FUNCTION_BLOCK RunUnitIndexerMasterCelluarA EXTENDS RunUnitIndexerMaster
VAR_INPUT
	// conveyor related , Fast + Slow = pitch
	ptCommandFast : POINTER TO CommandBlockPos;
	ptCommandSlow : POINTER TO CommandBlockPos;
	ptCommandExtend : POINTER TO CommandBlockPos;
	//Checkpoints
	ptCommandTriggerRaise: POINTER TO CommandBlockPos; //trigger point
	ptCommandCheckRaise : POINTER TO commandBlockPos; //if not all lifter done until then , stop conveyor motion
	ptCommandCheckReach : POINTER TO commandBlockPos;
	//Lifters
	lifters : ARRAY[1..3] OF POINTER TO RunLifterCelluar;
END_VAR
VAR_OUTPUT
END_VAR
VAR
	bFast : BOOL;
	bSlow : BOOL;
	bExtend : BOOL;
	
	nCounter  : INT ;
	allLifterDone : BOOL;
	allLifterReach: BOOL;
END_VAR

//implement state 3

SUPER^(); //run indexer master

//Buffer modes
ptAxisMaster^.ExecuteCommandBlock(ptBlock := ptCommandFast,
	Execute:= bFast,
	Done=>);
ptAxisMaster^.ExecuteCommandBlock(ptBlock := ptCommandSlow,
	Execute:= bSlow,
	Done=>);
ptAxisMaster^.ExecuteCommandBlock(ptBlock := ptCommandExtend,
	Execute:= bExtend,
	Done=>);

allLifterDone := TRUE; //reset
FOR nCounter:=1 TO 3 BY 1 DO
	lifters[nCounter]^.AsStopper(Execute:= ptAxisMaster^.PositionFeedback >= DWORD_TO_LREAL(ptCommandTriggerRaise^.COORDINATE/1000),
		Done=>,
		Error=>);
	allLifterDone := allLifterDone AND lifters[nCounter]^.AsStopper.Done; //collect overall result
END_FOR

//Before check point
ptAxisMaster^.ExecuteCommandBlock(ptBlock:=ptCommandSlow,
	Execute:=allLifterDone AND ptAxisMaster^.PositionFeedback < DWORD_TO_LREAL(ptCommandCheckRaise^.COORDINATE/1000),
	Done =>);
	
	
CASE SUPER^.state OF
	3:
	//reset pos command to zero
	bFast := TRUE; //start to go
	4:
	//until trigger raise reached , trigger all lifter to move
	IF ptAxisMaster^.PositionFeedback < DWORD_TO_LREAL(ptCommandCheckRaise^.COORDINATE/1000) THEN
		//transition
	END_IF
	5:
	//until check raise reached , check if all lifter done
	IF allLifterDone AND ptAxisMaster^.PositionFeedback < DWORD_TO_LREAL(ptCommandCheckRaise^.COORDINATE/1000) THEN
		//success transition
	ELSIF ptAxisMaster^.PositionFeedback < DWORD_TO_LREAL(ptCommandCheckRaise^.COORDINATE/1000) THEN
		//lifter comes error
	END_IF
	6: 
	// check reach
	IF allLifterReach AND ptAxisMaster^.PositionFeedback < DWORD_TO_LREAL(ptCommandCheckReach^.COORDINATE/1000) THEN
		//success transition
	ELSIF ptAxisMaster^.PositionFeedback >= DWORD_TO_LREAL(ptCommandCheckReach^.COORDINATE/1000) THEN
		//need walk further more	
	END_IF
	100:
	//any lifter fails , execute stop ( or not)
END_CASE

END_FUNCTION_BLOCK

(* stored: Version 1.1.0.1, ProductVersion 3.1.4020.12
   POU RunUnitIndexerMasterCelluarA: Id {8c290897-f573-4530-b2b8-1a75c3433cf9}, SpecialFunc None *)
